{attribute 'linkalways'}
{attribute 'no_explicit_call' := 'This FB is a CLASS and must be accessed using methods or properties'}
FUNCTION_BLOCK PUBLIC FileLogTargetAdapter IMPLEMENTS LogTargetAdapter
VAR CONSTANT
	message_buffer_capacity : UDINT := 100; // Number of messages that can be buffered
END_VAR
VAR
	// Configuration
	file_path : STRING := 'C:\';
	file_name : STRING := 'tclog.log';
	
	rolling_interval : RollingInterval := RollingInterval.Daily;
	/// When should old log files be deleted? Unit: days. Set it to `0` if log files should never be deleted. 
	log_lifespan : UINT := 0;
	timestamp_format : STRING := 'YYYYMMDD_hhmm_';

	log_cache : DynamicStringBuffer;
	date_time : DateTime;

	utc_time_as_file_time : Tc2_Utilities.T_FileTime; // Current utc time as filetime
	local_time_as_system_time : Tc2_Utilities.TimeStruct; // Current local time as timestring
	local_time_as_string : STRING; // Current local time as string

	formatter : DefaultFileLogEventFormatter;

	_error : Error; // Contains information about internal error.
	_busy : BOOL; // Logger is busy, typically with writing logs to the file system.
	
	rolling_interval_detector : RollingIntervalDetector;
	
	file_name_truncated : STRING;
	file_name_extension : STRING;
END_VAR

/// Configuration method which sets the lifespan of log files. Once exceeded, they will be deleted.
METHOD PUBLIC DeleteLogFilesAfterDays : REFERENCE TO FileLogTargetAdapter
VAR_INPUT
	/// Lifespan of logfiles in days.
	lifespan : UINT; 
END_VAR
log_lifespan := lifespan;

DeleteLogFilesAfterDays REF= THIS^;
END_METHOD

//FB_Init is always available implicitly and it is used primarily for initialization.
//The return value is not evaluated. For a specific influence, you can also declare the
//methods explicitly and provide additional code there with the standard initialization
//code. You can evaluate the return value.
METHOD FB_Init: BOOL
VAR_INPUT
    bInitRetains: BOOL; // TRUE: the retain variables are initialized (reset warm / reset cold)
    bInCopyCode: BOOL;  // TRUE: the instance will be copied to the copy code afterward (online change)   
END_VAR
log_cache.Init(message_buffer_capacity * (Tc2_System.Max_String_Length + Constants.FifoOverhead));
END_METHOD

/// Configuration method
/// Sets file_name of log file.
METHOD PUBLIC FileName : REFERENCE TO FileLogTargetAdapter
VAR_INPUT
	/// File name where the logs should be written to. Should not include path.
	file_name : STRING;
END_VAR
VAR
	last_period_index : INT;
END_VAR
THIS^.file_name := file_name;

last_period_index := FindLastOccurrence(file_name, '.');

IF last_period_index <> 0 THEN
	file_name_extension := GetFileExtension(file_name);
ELSE
	file_name_extension := 'log';
END_IF

FileName REF= THIS^;
END_METHOD

/// Configuration method
/// Sets file_path for log files.
METHOD PUBLIC FilePath : REFERENCE TO FileLogTargetAdapter
VAR_INPUT
	/// File path where the logs should be written to. Will be prefixed to `FileName`
	file_path : STRING; 
END_VAR
THIS^.file_path := file_path;

FilePath REF= THIS^;
END_METHOD

/// Flushes the logging cache. All messages that have not yet been processed will be lost.
METHOD PUBLIC FlushCache : BOOL
log_cache.FlushCache();
END_METHOD

METHOD PUBLIC Run
VAR_INST
	new_day : Tc2_Standard.R_Trig; 
	delete_expired_log_files : DeleteOldFiles;
	file_name_string_builder : StringBuilder;
	time_stamp : STRING; // Timestamp used for filename
	time_info_ready : BOOL := FALSE; // Set to true once the time information is available
	internal_error_occured : BOOL; // Aux variable to log internal errors to Error-property.
END_VAR
// Generate time data (shared state)
date_time.CyclicCall();
IF date_time.Done THEN
	time_info_ready := TRUE;
END_IF

local_time_as_system_time := date_time.AsLocalSystemTime;
local_time_as_string := date_time.AsLocalSystemTimeString;
utc_time_as_file_time := date_time.AsUtcFileTime;

rolling_interval_detector.Run(local_time_as_system_time);

// Generate new timestamp for filename
IF rolling_interval_detector.IntervalRolled(rolling_interval) OR date_time.Done THEN
	time_stamp := date_time.ToFormatString(timestamp_format);
END_IF

// Delete expired log files
new_day(Clk := local_time_as_system_time.wHour = 0);
delete_expired_log_files(
	StartScan 			:= 	new_day.Q AND (log_lifespan > 0),
	ExpirationInDays 	:=	log_lifespan,
	FilePath			:=	file_path,
	FileName 			:=	file_name,
	CurrentUtcTime 		:= 	utc_time_as_file_time	
);
IF delete_expired_log_files.Error.Active THEN
	internal_error_occured := TRUE;
	_error := delete_expired_log_files.Error;
END_IF
		
// Persist logging messages to file
log_cache.PersistToFile(
	time_info_ready,
	file_name_string_builder
		.Reset()
		.Append(file_path)
		.AppendIf(Tc2_Standard.Right(file_path, 1) <> '\', '\')
		.Append(time_stamp)
		.Append(file_name)
		.ToString()
);
IF log_cache.Error.Active THEN
	internal_error_occured := TRUE;
	_error := log_cache.Error;
END_IF

// Reset error flag each cycle to automatically confirm errors once they are gone.
IF NOT internal_error_occured THEN
	_error.Active := FALSE;
	_error.Code := ErrorCodes.None;
	_error.Info := '';
END_IF
internal_error_occured := FALSE;
END_METHOD

METHOD PUBLIC SendLogEvent : BOOL
VAR_INPUT
	event : LogEvent;
END_VAR
log_cache.AddLine(formatter.Format(event));
END_METHOD

/// Configuration method.
/// Sets the rolling interval of the log file. Once the rolling interval
/// expires, a file name with a new timestamp will be generated.
METHOD PUBLIC SetRollingInterval : REFERENCE TO FileLogTargetAdapter
VAR_INPUT
	/// Rolling interval for log file. Once exceeded, a new log file will be created.
	interval : RollingInterval; 
END_VAR
rolling_interval := interval;

SetRollingInterval REF= THIS^;
END_METHOD

END_FUNCTION_BLOCK

(* stored: Version 1.1.0.1
   POU FileLogTargetAdapter: Id {172ddd48-7f84-4661-9ada-761cf85c51a9}, SpecialFunc None
   Folder Configuration: Id {28a48266-87e4-495d-a151-e76531510359}
   Folder Constructor: Id {8be6375e-8e45-4885-bc59-a248a8bf47dc}
   Method DeleteLogFilesAfterDays: Id {32410822-67bd-4c13-a83d-53eb1112e24c}
   Method FB_Init: Id {5d0e415b-4d50-44cf-9e0d-7675377fd9fc}
   Method FileName: Id {6ad6fc1a-70ae-4fe8-a426-3bcf9a84e855}
   Method FilePath: Id {339d2aac-b7be-4a39-aa0b-4a5126dc4906}
   Method FlushCache: Id {37c75623-56f0-45e8-8045-828b74c5a501}
   Method Run: Id {ec75d489-513f-4f09-8e6c-6d2e82b7e0d2}
   Method SendLogEvent: Id {9b0ec506-83b0-4354-a8f0-2afcd94dd817}
   Method SetRollingInterval: Id {6b6a98f5-4ff4-49b0-80a7-0a8439a6af3a} *)
